ROGRAM p_Shakers
VAR
END_VAR

(* stored: Version 1.1.0.1, ProductVersion 3.1.4020.6
   POU p_Shakers: Id {017c063a-5f09-4d50-9c5d-ffc48aeba37a}, SpecialFunc None *)
